// TwinCAT 3 PLC project ScorerMisfeedPLC
// ProgramVersion: 3.1.4026.15
// libraries:
//   Tc2_Standard, * (Beckhoff Automation GmbH)
//   Tc2_System, * (Beckhoff Automation GmbH)
// project tree:
//   DUTs/ StateType.TcDUT
//   GVLs/ Global.TcGVL
//   / PlcTask.TcTTO
//   POUs/ MAIN.TcPOU
// real-time tasks:
//   TASK PlcTask: cycle T#10ms, priority 20, ADS port 350
// I/O:
//   DEVICE Device 1 (NOV-DP-RAM)
//   DEVICE Device 2 (Onboard I/O Device), AmsNetId 5.156.234.158.3.1
//     Term 1 (CX7028) [CX7028-0000-0121]
//       modules: Module 1 (DIO_2x), Module 2 (Empty Module), Module 3 (DIO_2x), Module 4 (Empty Module), Module 5 (DI_2x), Module 6 (Empty Module), Module 7 (DI_2x), Module 8 (Empty Module)
// variable links:
//   ScorerMisfeedPLC/ScorerMisfeedPLC Instance <-> Device 2 (Onboard I/O Device)/Term 1 (CX7028)
//     PlcTask Inputs/Global.bCoverFeedNoSheet <-> Module 3 (DIO_2x)/DIO_2x Input Channel 1/Input
//     PlcTask Inputs/Global.bCycleTrigger <-> Module 3 (DIO_2x)/DIO_2x Input Channel 2/Input
//     PlcTask Inputs/Global.bScorerCam <-> Module 1 (DIO_2x)/DIO_2x Input Channel 1/Input
//     PlcTask Inputs/Global.bScorerSheetDetected <-> Module 1 (DIO_2x)/DIO_2x Input Channel 2/Input
//     PlcTask Outputs/Global.bMisfeedAlarm <-> Module 1 (DIO_2x)/DIO_2x Output Channel 1/Output
//     PlcTask Outputs/Global.bMisfeedAlarm2 <-> Module 1 (DIO_2x)/DIO_2x Output Channel 2/Output

CONFIGURATION ScorerMisfeedPLC
    RESOURCE PLC ON TwinCAT3
        TASK PlcTask(INTERVAL := T#10ms, PRIORITY := 20);
        PROGRAM MAIN WITH PlcTask : MAIN;
    END_RESOURCE
END_CONFIGURATION

// ---- DUTs/StateType.TcDUT
{attribute 'qualified_only'}
{attribute 'strict'}
{attribute 'to_string'}

TYPE StateType :
(
	S0_SHEET_NOT_EXPECTED,
	S1_SHEET_SEARCH,
	S2_BREAK_SEARCH,
	S3_BREAK_COMPLETE,
	S4_CYCLE_COMPLETE,
	S8_FAULT
);
END_TYPE

// The back of the sheet is a predictable position.
// Small pulse first, then long pulse

// The sequence is
// - Cover should be present when short pulse positive edge
// - Then cover should have negative edge during long pulse

// No sheet expected
// Waiting for sheet
// - On cam positive edge check if the sheet is present
// Waiting for break
// - On

// ---- GVLs/Global.TcGVL
{attribute 'qualified_only'}
VAR_GLOBAL
	bScorerCam 					AT%I* :BOOL;
	bScorerSheetDetected		AT%I* :BOOL;
	bCoverFeedNoSheet		 	AT%I* :BOOL;
	bCoverSheetDetected		    	  :BOOL;
	bCycleTrigger 				AT%I* :BOOL;
	
	bMisfeedAlarm				AT%Q* :BOOL;
	bMisfeedAlarm2				AT%Q* :BOOL;
	
	stateHistory : ARRAY[1..32] OF INT;
END_VAR

// ---- POUs/MAIN.TcPOU
PROGRAM MAIN
VAR
	iCycleCount : INT;
	cycleTrigger : Tc2_Standard.R_TRIG;
	
	shiftRegister : WORD := 0;
	shiftInput : BOOL;
	
	coverFrontEdge : Tc2_Standard.R_TRIG;
	coverBackEdge : Tc2_Standard.F_TRIG;
	
	camFrontEdge : Tc2_Standard.R_TRIG;
	camBackEdge : Tc2_Standard.F_TRIG;
	
	state : StateType := StateType.S0_SHEET_NOT_EXPECTED;
	nextState : StateType := StateType.S0_SHEET_NOT_EXPECTED;
	first : BOOL := TRUE;
	
	resetTimer : TON;
	fault: BOOL := FALSE;
	
	flasher : TON;
	
	i : INT := 0;
	
	cycleCount : INT := 0;
	s121Count  : INT := 0; //should be 2x cycle count
END_VAR

// Every cycle we need to see if there is a cover sheet being loaded
// It takes 3 cycles for a cover sheet to get to the scorer
// If there is a cover sheet in the scorer we need to check
// 		- that there is a sheet there during the first pulse
//		- that there isn't a sheet present during the second pulse
// At all other times we shouldn't see a sheet in the scorer for either pulse

Global.bCoverSheetDetected := NOT Global.bCoverFeedNoSheet;

cycleTrigger(CLK := Global.bCycleTrigger);
coverFrontEdge(CLK := Global.bScorerSheetDetected);
coverBackEdge(CLK := Global.bScorerSheetDetected);
camFrontEdge(CLK := Global.bScorerCam);
camBackEdge(CLK := Global.bScorerCam);

resetTimer(IN := fault, PT := T#1S);
flasher(IN := NOT flasher.Q, PT := T#250MS);

IF cycleTrigger.Q THEN
	iCycleCount := iCycleCount + 1;
	shiftRegister := SHL(shiftRegister, 1);
	shiftRegister.0 := Global.bCoverSheetDetected;
END_IF;

CASE state OF
	StateType.S0_SHEET_NOT_EXPECTED:
		IF first THEN
			fault := FALSE;
		END_IF
		
		IF shiftRegister.1 THEN
			nextState := StateType.S1_SHEET_SEARCH;                   // S0 -> S1
		ELSIF coverFrontEdge.Q AND NOT shiftRegister.0 THEN
			nextState := StateType.S8_FAULT;                          // S0 -> S8
		END_IF
		
	StateType.S1_SHEET_SEARCH:
		IF camFrontEdge.Q THEN
			IF Global.bScorerSheetDetected THEN
				nextState := StateType.S2_BREAK_SEARCH;               // S1 -> S2
			ELSE
				nextState := StateType.S8_FAULT;                      // S1 -> S8
			END_IF
		END_IF
		
	StateType.S2_BREAK_SEARCH:
		IF camFrontEdge.Q THEN
			IF NOT Global.bScorerSheetDetected THEN
				nextState := StateType.S3_BREAK_COMPLETE;             // S2 -> S3
			ELSE
				nextState := StateType.S8_FAULT;                      // S2 -> S8
			END_IF
		END_IF
	
	StateType.S3_BREAK_COMPLETE:
		IF camBackEdge.Q THEN
			IF NOT Global.bScorerSheetDetected THEN
				nextState := StateType.S4_CYCLE_COMPLETE;             // S3 -> S4
			ELSE
				nextState := StateType.S8_FAULT;                      // S3 -> S8
			END_IF
		END_IF
	
	StateType.S4_CYCLE_COMPLETE:
		IF cycleTrigger.Q THEN
			nextState := StateType.S0_SHEET_NOT_EXPECTED;             // S4 -> S0
		END_IF
		
	StateType.S8_FAULT:
		Global.bMisfeedAlarm := TRUE;
		fault := TRUE;
		IF flasher.Q THEN
			Global.bMisfeedAlarm2 := TRUE;
		ELSE
			Global.bMisfeedAlarm2 := FALSE;
		END_IF
		IF resetTimer.Q THEN
			Global.bMisfeedAlarm := FALSE;
			Global.bMisfeedAlarm2 := FALSE;
			nextState := StateType.S4_CYCLE_COMPLETE;
			ADSLOGSTR(msgCtrlMask := ADSLOG_MSGTYPE_STRING, msgFmtStr := 'S8 -> S4', strArg := '');
		END_IF
END_CASE

IF cycleTrigger.Q THEN
	cycleCount := cycleCount + 1;
END_IF

IF camFrontEdge.Q THEN
	s121Count := s121Count + 1;
END_IF


IF state <> nextState THEN
	first := TRUE;
	state := nextState;
	FOR i := 32 TO 2 BY -1 DO
		Global.stateHistory[i] := Global.stateHistory[i - 1];
	END_FOR
	Global.stateHistory[1] := state;
ELSE
	first := FALSE;
END_IF

END_PROGRAM
